PROGRAM Grabber_Timeout
VAR
END_VAR

Timers.GrabberClosing[1](IN:= Shuttle.GrabberIsClosing[1], PT:= T#5S, Q=> , ET=> );
Timers.GrabberClosing[2](IN:= Shuttle.GrabberIsClosing[2], PT:= T#5S, Q=> , ET=> );

Timers.GrabberOpening[1](IN:= Shuttle.GrabberIsOpening[1], PT:= T#5S, Q=> , ET=> );
Timers.GrabberOpening[2](IN:= Shuttle.GrabberIsOpening[2], PT:= T#5S, Q=> , ET=> );

IF Timers.GrabberClosing[1].Q THEN
	
	Shuttle.OpenFaultedGrabber[1]		:= TRUE;
	Shuttle.GrabberFaulted[1]			:= TRUE;
		
END_IF

IF Timers.GrabberClosing[2].Q THEN
	
	Shuttle.OpenFaultedGrabber[2]		:= TRUE;
	Shuttle.GrabberFaulted[2]			:= TRUE;
		
END_IF

IF Timers.GrabberOpening[1].Q THEN
	
	Shuttle.CloseFaultedGrabber[1]		:= TRUE;
	Shuttle.GrabberFaulted[1]			:= TRUE;
		
END_IF

IF Timers.GrabberOpening[1].Q THEN
	
	Shuttle.CloseFaultedGrabber[1]		:= TRUE;
	Shuttle.GrabberFaulted[2]			:= TRUE;
		
END_IF

IF Shuttle.Reset THEN

	Shuttle.GrabberFaulted[1]			:= FALSE;
	Shuttle.GrabberFaulted[2]			:= FALSE;	
	Shuttle.OpenFaultedGrabber[1] 		:= FALSE;
	Shuttle.OpenFaultedGrabber[2]		:= FALSE;
	Shuttle.CloseFaultedGrabber[1]		:= FALSE;
	Shuttle.CloseFaultedGrabber[2]		:= FALSE;
	
END_IF

IF Shuttle.CloseFaultedGrabber[1] THEN
	
	Close_Grabber_1();

END_IF

IF Shuttle.CloseFaultedGrabber[2] THEN
	
	Close_Grabber_2();

END_IF

IF Shuttle.OpenFaultedGrabber[1] THEN
	
	Open_Grabber_1();

END_IF

IF Shuttle.OpenFaultedGrabber[2] THEN
	
	Open_Grabber_2();

END_IF

END_PROGRAM

(* stored: Version 1.1.0.1, ProductVersion 3.1.4024.9
   POU Grabber_Timeout: Id {6d28266a-e721-4911-a9eb-af5e3c5ad838}, SpecialFunc None *)
